# EPICS substitutions: ek9000App/Db/EL1702.substitutions
file EL1702.template
{       pattern
        {
                TERMINAL,

        }
        {
        }
}
